(* IEC 61131-3 sources: axopen.templates/axopen.template.simple/ax/src/templates/starterunit/Modes, 3 files *)

(* ---- AutomatSequence.st ---- *)
NAMESPACE axosimple.StarterUnitTemplate
    USING axosimple;
    USING AXOpen.Data;
    USING AXOpen.Core;
    USING System.Strings;

    ///<summary>
    /// Provides automatic mode sequence for `StarterUnitTemplate` unit.
    ///</summary>
    {#ix-set:AttributeName = "<#AUTOMAT#>"}
    {S7.extern=ReadWrite}
    CLASS PUBLIC AutomatSequence
        EXTENDS AXOpen.Core.AxoSequencerContainer IMPLEMENTS IModeContainer
        VAR PUBLIC
            ///<summary>
            /// Step coordinators for this sequence.
            ///</summary>
            Steps : ARRAY[0..100] OF AxoStep;

            _inspectionResult: BOOL;
            _inspectionValue: LREAL;
            _inspectionData: STRING;

            _comprehensiveResult: AXOpen.Inspectors.AxoComprehensiveResult;
        END_VAR

        VAR PRIVATE
            X : REF_TO axosimple.StarterUnitTemplate.UnitObjects;

            _currentId : STRING;

            _dialogAnswer : eDialogAnswer;
            _externalCloseOkSignal : BOOL;
        END_VAR

        METHOD INTERNAL Run
            VAR_INPUT
                inParent : AXOpen.Core.IAxoObject;
                inUnitObjects : REF_TO UnitObjects;
            END_VAR

            IF X = NULL THEN
                X := inUnitObjects;
            END_IF;

            SUPER.Run(inParent);
        END_METHOD

        VAR
            resutl : IAxoTaskState;
            _isDone : BOOL;
        END_VAR

        METHOD PROTECTED OVERRIDE OnBeforeSequenceStart
            X^._inspectorDialog.Restore();
            X^.PD.Restore();
            X^.TD.Restore();
        END_METHOD

        ///<summary>
        ///     Contains logic of the steps of this sequence
        ///</summary>
        METHOD OVERRIDE Main
            VAR

            END_VAR

            IF (X = NULL) THEN
                RETURN;
            END_IF;

            // This sequecner executes the steps in cycles from top to bottom
            // in the same order they are written in the program
            // Each step in the sequence must can be used only once.
            // This sets the sequence to run in cycles (top-botton-top and again).
            THIS.SequenceMode := eAxoSequenceMode#Cyclic;

            IF (Steps[0].Execute(THIS, TRUE, '<#LOAD TECHNOLOGY DATA#>')) THEN
                //-------------------------------------------------------
                    IF(X^.TD.Read('default').IsDone()) THEN
                        THIS.MoveNext();
                    END_IF;
                //-------------------------------------------------------
            END_IF;

            IF (Steps[1].Execute(THIS, TRUE, '<#LOAD PROCESS DATA#>')) THEN
                //-------------------------------------------------------
                    IF(X^.PD.Read('default').IsDone()) THEN
                        _currentId := ToString(THIS.GetContext().GetRtc().NowUTC());
                        THIS.MoveNext();
                    END_IF;
                //-------------------------------------------------------
            END_IF;

            IF (Steps[2].Execute(THIS, TRUE, CONCAT('CREATE ITEM: ',_currentId))) THEN
                //-------------------------------------------------------

                IF (X^.PD.CreateOrUpdate(_currentId).IsDone()) THEN
                    THIS.MoveNext();
                END_IF;
                //-------------------------------------------------------
            END_IF;

            IF (Steps[3].Execute(THIS, TRUE, '<#Dialog notify#>')) THEN
                //-------------------------------------------------------
                //_externalCloseOkSignal := CurrentStep.Duration > dialogTimeOut;

                _dialogAnswer := X^._dialog.ShowWithExternalClose(THIS, _externalCloseOkSignal)
                .WithOK()
                .WithType(eDialogType#Info)
                .WithCaption('Info caption!')
                .WithText('Info - dialog will be closed by external timeout 2s!').Answer();

                IF( _dialogAnswer = eDialogAnswer#Ok) THEN
                    THIS.MoveNext();
                END_IF;
                //-------------------------------------------------------
            END_IF;

            IF (Steps[4].Execute(THIS, TRUE, '<#Dialog success#>')) THEN
                //-------------------------------------------------------
                //_externalCloseOkSignal := CurrentStep.Duration > dialogTimeOut;

                    _dialogAnswer := X^._dialog.ShowWithExternalClose(THIS, _externalCloseOkSignal)
                    .WithOK()
                    .WithType(eDialogType#Success)
                    .WithCaption('Success caption!')
                    .WithText('Success - dialog will be closed by external timeout 2s!').Answer();

                    IF( _dialogAnswer = eDialogAnswer#Ok) THEN
                        THIS.MoveNext();
                    END_IF;
                //-------------------------------------------------------
            END_IF;

            IF (Steps[5].Execute(THIS, TRUE, '<#Dialog Warning#>')) THEN
                //-------------------------------------------------------
                //_externalCloseOkSignal := CurrentStep.Duration > dialogTimeOut;

                    _dialogAnswer := X^._dialog.ShowWithExternalClose(THIS, _externalCloseOkSignal)
                    .WithYesNo()
                    .WithType(eDialogType#Warning)
                    .WithCaption('Warning caption!')
                    .WithText('Warning - dialog will be closed by external timeout 2s!').Answer();

                    IF( _dialogAnswer = eDialogAnswer#Yes) THEN
                        THIS.MoveNext();
                    END_IF;
                //-------------------------------------------------------
            END_IF;

            IF (Steps[6].Execute(THIS, TRUE, '<#Dialog danger#>')) THEN
                //-------------------------------------------------------
                //_externalCloseOkSignal := CurrentStep.Duration > dialogTimeOut;

                    _dialogAnswer := X^._dialog.ShowWithExternalClose(THIS, _externalCloseOkSignal)
                    .WithYesNoCancel()
                    .WithType(eDialogType#Warning)
                    .WithCaption('Danger caption!')
                    .WithText('Danger - dialog will be closed by external timeout 2s!').Answer();

                    IF( _dialogAnswer = eDialogAnswer#Yes) THEN
                        THIS.MoveNext();
                    END_IF;
                //-------------------------------------------------------
            END_IF;

            IF (Steps[7].Execute(THIS, TRUE, 'Example Digital inspection')) THEN
                //-------------------------------------------------------
                X^.PD.Data.Payload.PartPresence.WithCoordinator(THIS).Inspect(THIS,_inspectionResult)
                .UpdateComprehensiveResult(_comprehensiveResult)
                .OnFail()
                .CarryOn();
                //-------------------------------------------------------
            END_IF;

            IF (Steps[8].Execute(THIS, TRUE, 'Example Analog inspection')) THEN
                //-------------------------------------------------------
                _inspectionValue := -5500;

                X^.PD.Data.Payload.LoadPosition.WithCoordinator(THIS)
                .Inspect(THIS,_inspectionValue)
                .UpdateComprehensiveResult(_comprehensiveResult)
                .OnFail()
                .Dialog( inRetryStep := Steps[50], inTerminateStep := Steps[60], inoDialog := X^._inspectorDialog);
                //-------------------------------------------------------
            END_IF;

            IF (Steps[9].Execute(THIS, TRUE, 'Example Data inspection')) THEN
                //-------------------------------------------------------
                _inspectionData := 'tempCode';

                X^.PD.Data.Payload.JigDataMatrixCode.WithCoordinator(THIS)
                .Inspect(THIS,_inspectionData)
                .UpdateComprehensiveResult(_comprehensiveResult)
                .OnFail()
                .Dialog( inRetryStep := Steps[70], inTerminateStep := Steps[80], inoDialog := X^._inspectorDialog);
                //-------------------------------------------------------
            END_IF;

            IF (Steps[99].Execute(THIS, TRUE,CONCAT('UPDATE ITEM: ', _currentId))) THEN
                //-------------------------------------------------------
                IF (X^.PD.Update(_currentId).IsDone()) THEN
                    THIS.MoveNext();
                END_IF;
                //-------------------------------------------------------
            END_IF;

            // This will close the sequence and will return to the first step.
            THIS.Close(Steps[100]);
        END_METHOD
    END_CLASS

END_NAMESPACE

(* ---- GroundSequence.st ---- *)
NAMESPACE axosimple.StarterUnitTemplate
    USING axosimple;
    USING AXOpen.Data;
    USING AXOpen.Core;
    USING System.Strings;

    ///<summary>
    /// Provides ground mode sequence.
    ///</summary>
    {#ix-set:AttributeName = "<#GROUND#>"}
    {S7.extern=ReadWrite}
    CLASS PUBLIC GroundSequence
        EXTENDS AXOpen.Core.AxoSequencerContainer IMPLEMENTS IModeContainer
        VAR PUBLIC
            Steps : ARRAY[0..100] OF AXOpen.Core.AxoStep;
            MoveToWork : AXOpen.Core.AxoTask;
        END_VAR
        VAR PRIVATE
            X : REF_TO axosimple.StarterUnitTemplate.UnitObjects;
            PersistentSettings : REF_TO AxoDataPersistentExchange;
            _currentId : STRING;
            techSetttingsId : STRING;
        END_VAR

        METHOD INTERNAL Run
            VAR_INPUT
                inParent : AXOpen.Core.IAxoObject;
                inUnitObjects : REF_TO axosimple.StarterUnitTemplate.UnitObjects;
            END_VAR

            IF X = NULL THEN
                X := inUnitObjects;
                PersistentSettings := X^.G^.Persits;
            END_IF;

            SUPER.Run(inParent);
        END_METHOD

        METHOD PROTECTED OVERRIDE OnBeforeSequenceStart
            X^.TD.Restore();
            X^.PD.Data.Restore();
            X^._DL.Restore();
            X^._ADL.Restore();
            X^._IDL.Restore();
        END_METHOD

        ///<summary>
        /// Contains logic of the steps of this sequence
        ///</summary>
        METHOD PROTECTED OVERRIDE Main
            VAR
                taskState : AXOpen.Core.IAxoTaskState;
                forIterator : INT;
                _dialogAnswer : eDialogAnswer;
            END_VAR;
            // IF (Components = NULL OR ProcessData = NULL) THEN
            //     RETURN;
            // END_IF;
            // This sequecner executes the steps in cycles from top to bottom
            // in the same order they are written in the program
            // Each step in the sequence must can be used only once.
            // This sets the sequence to run once (top-botton) and stops with done after closing.
            THIS.SequenceMode := eAxoSequenceMode#RunOnce;

            IF (Steps[0].Execute(THIS, TRUE, '<#DIALOG#>')) THEN
                //-------------------------------------------------------

                _dialogAnswer := X^._DL.Show(THIS).WithCaption('<#DO YOU WANT TO RUN THE GROUND MODE SEQUENCE?#>').WithYesNo().WithType(eDialogType#Warning).Answer();

                IF(_dialogAnswer <> eDialogAnswer#NoAnswer) THEN
                    IF(_dialogAnswer = eDialogAnswer#Yes) THEN
                        THIS.MoveNext();
                    END_IF;

                    IF(_dialogAnswer = eDialogAnswer#No) THEN
                        THIS.Restore();
                    END_IF;
                END_IF;
                //-------------------------------------------------------
            END_IF;

            // This is more verbose but also more versatile way of executing step logic.
            IF (Steps[1].Execute(THIS, TRUE, '<#RESTORE#>')) THEN
                //-------------------------------------------------------
                IF(X <> NULL) THEN
                    X^.TD.Restore();
                    X^.PD.Data.Restore();
                    X^._DL.Restore();
                    X^._ADL.Restore();
                    X^._IDL.Restore();
                    THIS.MoveNext();
                END_IF;
                //-------------------------------------------------------
            END_IF;

            IF (Steps[2].Execute(THIS, TRUE, '<#READ PERSISTENT SETTINGS#>')) THEN
                //-------------------------------------------------------
                IF CurrentStep.IsFirstEntryToStep() THEN
                    ;// some special initialization
                END_IF;

                CASE TO_INT( THIS.GetMicroStepValue()) OF
                    0 :
                        IF PersistentSettings^.InvokeEntityExist(THIS ,'') THEN
                            THIS.SetMicroStepValue(UINT#10);
                        END_IF;

                    10 :
                        IF PersistentSettings^.IsEntityExistDone(THIS) THEN
                            IF PersistentSettings^.EntityExistResult() THEN
                                THIS.SetMicroStepValue(UINT#40); // default data exist
                            ELSE
                                THIS.SetMicroStepValue(UINT#20); // no data exist
                            END_IF;
                        END_IF;

                    20 :
                        IF PersistentSettings^.InvokeUpdateAll(THIS) THEN // data not exist -> udate all to DB
                            THIS.SetMicroStepValue(UINT#30);
                        END_IF;

                    30:
                        IF PersistentSettings^.IsUpdateAllDone(THIS) THEN
                            THIS.SetMicroStepValue(UINT#40); // all was updated to DB
                        END_IF;

                    40 :
                        IF PersistentSettings^.InvokeRead(THIS, '') THEN // read default group
                            THIS.SetMicroStepValue(UINT#50);
                        END_IF;
                    50 :
                        IF PersistentSettings^.IsReadDone(THIS) THEN
                                THIS.MoveNext(); // just default group was readed
                        END_IF;
                    ELSE
                        THIS.SetMicroStepValue(UINT#0);
                END_CASE;

                //-------------------------------------------------------
            END_IF;

            IF (Steps[5].Execute(THIS, TRUE, '<#READ TECHNOLOGY SETTINS#>')) THEN
                //-------------------------------------------------------

                IF CurrentStep.IsFirstEntryToStep() THEN
                    IF(X^.G = NULL) THEN RETURN; END_IF;
                    IF(X^.G^.TS = NULL) THEN RETURN; END_IF;

                    IF X^.G^.TS^.Common.Payload.DataEntityId <> '' THEN
                       techSetttingsId := X^.G^.TS^.Common.Payload.DataEntityId; // TAKE GLOGAL TECHNOLOGY SETTINGS ID

                    ELSIF X^.TD.Data.Payload.DataEntityId <> '' THEN // TAKE LAST LOADED FOR STATION
                        techSetttingsId := X^.TD.Data.Payload.DataEntityId;

                    ELSIF X^.LastTechnologySettings <> '' THEN // TAKE LAST LOADED FROM PERSISTENT
                        techSetttingsId := X^.LastTechnologySettings;
                    ELSE
                        X^.LastTechnologySettings := 'default'; // FORCE DEFAULT VALUE
                        techSetttingsId := X^.LastTechnologySettings;
                    END_IF;

                    IF X^.G^.TS^.Common.Payload.DataEntityId = X^.TD.Data.Payload.DataEntityId then
                        //THIS.MoveNext(); // you can skip loading...
                        ;
                    end_if;

                else
                    // IF(Objs^.TechnologySettings^.Read( techSetttingsId ).IsDone()) THEN
                    //     THIS.MoveNext();
                    // END_IF;
                    THIS.MoveNext();
                END_IF;
                //-------------------------------------------------------
            END_IF;

            FOR forIterator := 6 TO 98 BY 1 DO
                IF (Steps[forIterator].Execute(THIS, TRUE,Concat('DO SOMETHING -G-',ToString(forIterator)) )) THEN
                    //-------------------------------------------------------
                    IF CurrentStep.Duration > TIME#25ms THEN
                        THIS.MoveNext();
                    END_IF;
                    //-------------------------------------------------------
                END_IF;
            END_FOR;

            IF (Steps[99].Execute(THIS, TRUE, '<#SAVE DATA#>')) THEN
                //-------------------------------------------------------
                CASE TO_INT( THIS.GetMicroStepValue()) OF
                    0 :
                        IF X^.PD.Shared.Payload.DataEntityId <> '' THEN
                            _currentId := X^.PD.Shared.Payload.DataEntityId;
                            THIS.SetMicroStepValue(UINT#10);

                        ELSE // FIST RUN OR WITHOUT DATA
                            THIS.MoveNext();
                        END_IF;

                    10 : // update part as a corrupted a interrupted
                        X^.PD.Shared.Payload.WasReset := true;
                        IF X^.PD.Update(_currentId).IsDone() THEN
                                THIS.MoveNext();
                        END_IF;
                    ELSE
                        THIS.SetMicroStepValue(UINT#0);
                END_CASE;
                //-------------------------------------------------------
            END_IF;

            // This will close the sequence and will return to the first step.
            THIS.Close(Steps[100]);
        END_METHOD
    END_CLASS
END_NAMESPACE

(* ---- ServiceMode.st ---- *)
NAMESPACE axosimple.StarterUnitTemplate
    USING axosimple;
    USING AXOpen.Data;
    USING AXOpen.Core;
    USING System.Strings;

    ///<summary>
    /// Provides logic for service/manual/maintenance mode.
    ///</summary>
    {#ix-set:AttributeName = "<#SERVICE#>"}
    {S7.extern=ReadWrite}
    CLASS PUBLIC ServiceMode
        EXTENDS AXOpen.Core.AxoTask IMPLEMENTS IModeContainer
        ///<summary>
        /// Runs service mode logic. This method must be called cyclically.
        ///</summary>

        METHOD PUBLIC Run
            VAR_INPUT
                parent : IAxoObject;
            END_VAR
            VAR_IN_OUT
                C : axosimple.StarterUnitTemplate.Components;
            END_VAR
            THIS.Initialize(parent);
            IF THIS.Execute() THEN
                THIS.Handle(C);
            END_IF;
        END_METHOD

        METHOD PRIVATE Handle
            VAR_IN_OUT
                C : axosimple.StarterUnitTemplate.Components;
            END_VAR
            ;
            // HERE CALL LOGIC FOR MANUAL/SERICE OPERATIONS
        END_METHOD
    END_CLASS
END_NAMESPACE
